// Mitsubishi GX Works2 project: 241129_ex6   PLC: Q02U

PROGRAM MAIN
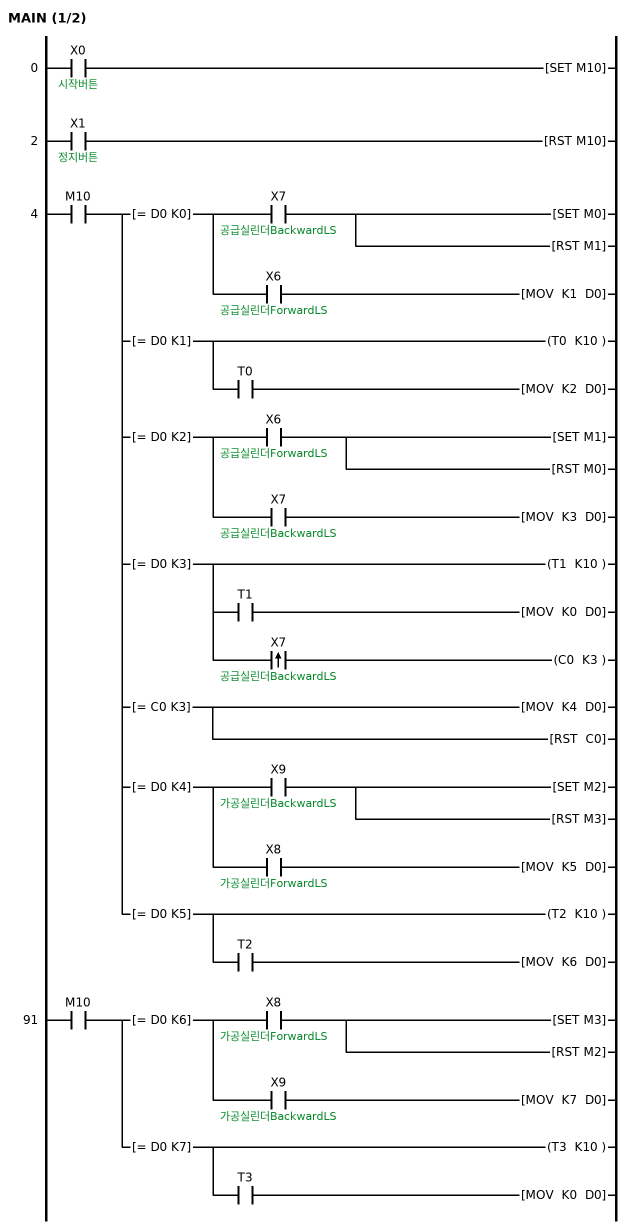
0     LD      X0  ; 시작버튼
      SET     M10
2     LD      X1  ; 정지버튼
      RST     M10
4     LD      M10
      MPS
      AND=    D0 K0
      MPS
      AND     X7  ; 공급실린더BackwardLS
      SET     M0
      RST     M1
      MPP
      AND     X6  ; 공급실린더ForwardLS
      MOV     K1 D0
      MRD
      AND=    D0 K1
      OUT     T0 K10
      AND     T0
      MOV     K2 D0
      MRD
      AND=    D0 K2
      MPS
      AND     X6  ; 공급실린더ForwardLS
      SET     M1
      RST     M0
      MPP
      AND     X7  ; 공급실린더BackwardLS
      MOV     K3 D0
      MRD
      AND=    D0 K3
      OUT     T1 K10
      MPS
      AND     T1
      MOV     K0 D0
      MPP
      ANDP    X7  ; 공급실린더BackwardLS
      OUT     C0 K3
      MRD
      AND=    C0 K3
      MOV     K4 D0
      RST     C0
      MRD
      AND=    D0 K4
      MPS
      AND     X9  ; 가공실린더BackwardLS
      SET     M2
      RST     M3
      MPP
      AND     X8  ; 가공실린더ForwardLS
      MOV     K5 D0
      MPP
      AND=    D0 K5
      OUT     T2 K10
      AND     T2
      MOV     K6 D0
91    LD      M10
      MPS
      AND=    D0 K6
      MPS
      AND     X8  ; 가공실린더ForwardLS
      SET     M3
      RST     M2
      MPP
      AND     X9  ; 가공실린더BackwardLS
      MOV     K7 D0
      MPP
      AND=    D0 K7
      OUT     T3 K10
      AND     T3
      MOV     K0 D0
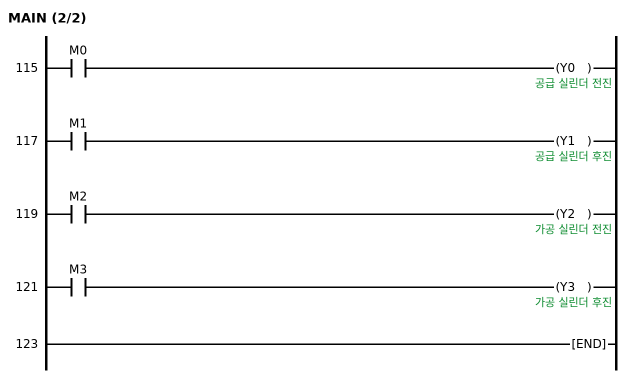
115   LD      M0
      OUT     Y0  ; 공급 실린더 전진
117   LD      M1
      OUT     Y1  ; 공급 실린더 후진
119   LD      M2
      OUT     Y2  ; 가공 실린더 전진
121   LD      M3
      OUT     Y3  ; 가공 실린더 후진
123   END
END_PROGRAM

// device comments not shown above
X2  ; 긴급정지버튼
X3  ; 공급센서
X4  ; 물체확인센서
X5  ; 금속확인센서
X0A  ; 송출실린더ForwardLS
X0B  ; 송출실린더BackwardLS
X0C  ; 배출실린더ForwardLS
X0D  ; 배출실린더BackwardLS
Y4  ; 송출 실린더 전진
Y5  ; 송출 실린더 후진
Y6  ; 배출 실린더 전진
Y7  ; 배출 실린더 후진
Y8  ; 컨베이어 CW
Y9  ; 컨베이어 CCW
Y0A  ; 컨베이어 STOP
Y0B  ; 램프 RED
Y0C  ; 램프 YELLOW
Y0D  ; 램프 GREEN
